{attribute 'qualified_only'}
{attribute 'strict'}
TYPE eCyclinderBaseTests : (
    Invalid := 50,
    GetAtHome := 100,
    GetAtWork := 200
);
END_TYPE

(* stored: Version 1.1.0.1, ProductVersion 3.1.4024.6
   DUT eCyclinderBaseTests: Id {bb45d148-104b-0e48-2d7d-958318741966} *)
